PROGRAM p_EtherCATDiag
VAR
    fbEcatDiag1	:	LCLS_General.FB_EcatDiag;
END_VAR

fbEcatDiag1(i_AMSNetId:=g_aEcatMaster1, i_xFirstPass:=g_xFirstPass, q_xAllStatesGood=>g_xIOState);

END_PROGRAM

(* stored: Version 1.1.0.1, ProductVersion 3.1.4020.14
   POU p_EtherCATDiag: Id {19e5e726-066d-4fae-968d-98c55136430e}, SpecialFunc None *)
